FUNCTION_BLOCK AutoSamplar_HMI (* Service Interface Function Block Type *)
  (* Standard: 61499-2 *)
  (* Version 0.0, 9/26/2024, SESA713705, Schneider Electric, template *)
  PACKAGE SE.Nereda;
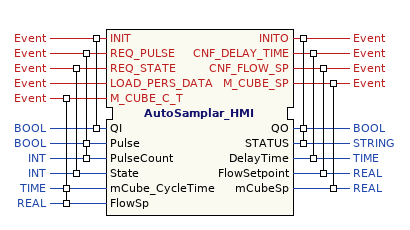
  EVENT_INPUT
    INIT WITH QI;
    REQ_PULSE WITH Pulse, PulseCount;
    REQ_STATE WITH State;
    LOAD_PERS_DATA;
    M_CUBE_C_T WITH mCube_CycleTime, FlowSp;
  END_EVENT
  EVENT_OUTPUT
    INITO WITH QO, STATUS;
    CNF_DELAY_TIME WITH DelayTime;
    CNF_FLOW_SP WITH FlowSetpoint;
    M_CUBE_SP WITH mCubeSp;
  END_EVENT
  VAR_INPUT
    QI : BOOL;
    Pulse : BOOL;
    PulseCount : INT;
    State : INT;
    mCube_CycleTime : TIME;
    FlowSp : REAL;
  END_VAR
  VAR_OUTPUT
    QO : BOOL; (* Event Output Qualifier *)
    STATUS : STRING; (* Service Status *)
    DelayTime : TIME;
    FlowSetpoint : REAL;
    mCubeSp : REAL;
  END_VAR
  SERVICE /
    SEQUENCE 
    END_SEQUENCE
  END_SERVICE
END_FUNCTION_BLOCK
